KUKA KRL program: chk_w11_grp3_clo.src

&ACCESS RVO3
&COMMENT Axor 913 Z3.1
DEF chk_w11_grp3_clo( )
; Check gripper AXOR 913 CLOSE Z3.1
;//---- Start User-------

$TIMER[10] = 0
$TIMER_STOP[10] = FALSE

WAIT FOR ($IN[534])
WAIT FOR (NOT $IN[533])

$TIMER_STOP[10] = TRUE
$TIMER[10] = 0

;//---- End User---------
END
